// TIA Portal V20 export
FUNCTION "DemoIdentRf" : Void   // FC79, LAD
TITLE = Demo: IDENT_FC / Demo: Ident
AUTHOR : SICAR
FAMILY : Demo
VERSION : 1.0
// Demo fuer Anwendung Ident Bausteine / Demo for usage of ident moduls
// stored: IsIECCheckEnabled true, SetENOAutomatically true
   // Ret_Val : Ret_Val
BEGIN

REGION Network 1: Änderungshistorie / ChangeLog
   // Die Änderungshistorie wird nur in englischer Editiersprache geführt.
   // Change log table:
   // Version | Date | Expert in charge | Changes applied
   // -------|---------|-------------|--------------------------------------------
   // 05.00.00 | 01.09.2023 | SICAR | First released version
END_REGION

REGION Network 2: Schreiben reader 1 / Define reading informations
   // Schreibe den String "Siemens" in die zu schreibende Datenstrucktur des RFID Geräts / Write the String "Siemens" in the writting structur of the FB
END_REGION

REGION Network 3: Schreiben reader 1 / Define writting informations
   // Schreibe den String "Siemens" in die zu schreibende Datenstrucktur des RFID Geräts / Write the String "Automation Framework" in the writting structur of the FB
END_REGION

REGION Network 4: Schreiben reader 1 / Define reading informations
   // Schreibe den String "Siemens" in die zu schreibende Datenstrucktur des RFID Geräts / Write the String "RF2385-621863" in the writting structur of the FB
END_REGION

REGION Network 5: Schreiben reader 1 / Define reading informations
   // Schreibe den String "Siemens" in die zu schreibende Datenstrucktur des RFID Geräts / Write the String "Demo RFID" in the writting structur of the FB
END_REGION
END_FUNCTION
